Universal Robots PolyScope program: vg_transpor_cards.urp

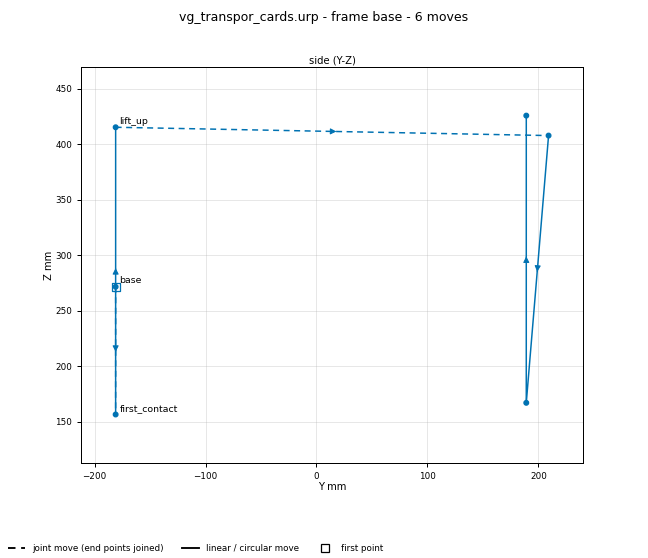
[picture p0: tool path of vg_transpor_cards.urp in frame base, 6 of 6 moves have a stored position in this frame; points joined in program order, loops and branches not executed]
Program vg_transpor_cards (installation=default directory=/programs/v_gripper_tm1326 createdIn=5.11.9.1010452 lastSavedIn=5.11.9.1010452 robotSerialNumber=20225200364)
Calibrated DH parameters: a=[0.00002, -0.569483, -0.54992, -0.00001, -0.000036, 0]; d=[0.180894, -146.691669, 192.918669, -46.053088, 0.119778, 0.115602]; alpha=[1.571425, -0.001534, 0.003359, 1.568739, -1.571477, 0]; deltaTheta=[0, 0.376258, -0.101074, -0.275185, -0.000002, 0]
Robot Program (runOnlyOnce=false)
  MoveJ speed 60 deg/s, acceleration 80 deg/s^2 (useActiveTCP=true) feature=Base
    Waypoint base: TCP in base x=421.909 y=-180.993 z=271.627 mm, rx=2.2364 ry=-2.2063 rz=0 rad; joints [-0.977, -80.029, -144.027, -45.908, 90.179, -1.705] deg
  MoveJ speed 60 deg/s, acceleration 80 deg/s^2 (useActiveTCP=true) feature=Base
    Waypoint first_contact: TCP in base x=421.917 y=-180.997 z=156.56 mm, rx=2.2364 ry=-2.2063 rz=-0.0001 rad; joints [-0.995, -95.96, -149.103, -24.902, 90.113, -1.657] deg
    URCap VG Grip (OnRobot, OnRobot A/S) dataModel(vg.grip.target.vacuum=5000.0, Variable(key=on_return, variable(name=on_return)))
  MoveL speed 250 mm/s, acceleration 1200 mm/s^2 (useActiveTCP=true) feature=Base
    Waypoint lift_up: TCP in base x=421.921 y=-180.985 z=415.39 mm, rx=2.2364 ry=-2.2063 rz=0 rad; joints [-0.961, -68.742, -134.04, -67.181, 90.213, -1.769] deg
  MoveJ speed 60 deg/s, acceleration 80 deg/s^2 (useActiveTCP=true) feature=Base
    Waypoint above_des: TCP in base x=421.893 y=209.131 z=407.905 mm, rx=2.2364 ry=-2.2062 rz=0 rad; joints [48.034, -70.642, -133.728, -65.599, 90.214, 47.234] deg
  MoveL speed 250 mm/s, acceleration 1200 mm/s^2 (useActiveTCP=true) feature=Base
    Waypoint before_dropping: TCP in base x=424.684 y=189.04 z=167.078 mm, rx=2.2365 ry=-2.2062 rz=-0.0001 rad; joints [45.929, -94.755, -148.182, -27.028, 90.123, 45.255] deg
    URCap VG Release (OnRobot, OnRobot A/S)
    Waypoint up_from_des: TCP in base x=424.683 y=189.058 z=425.891 mm, rx=2.2365 ry=-2.2061 rz=-0.0001 rad; joints [45.961, -68.974, -132.767, -68.227, 90.22, 45.146] deg
    Halt
